// Mitsubishi GX Developer project: continuous   PLC: FX3U

PROGRAM MAIN
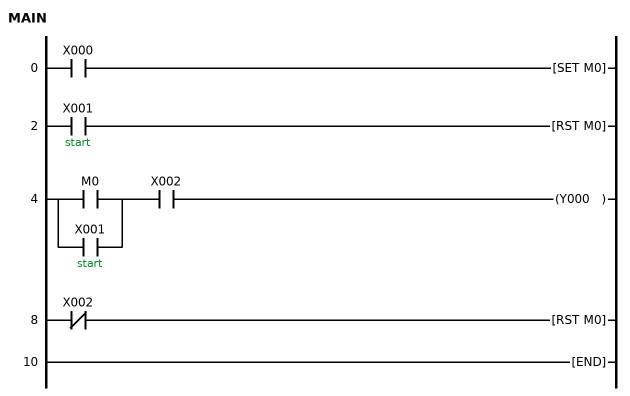
0     LD      X000
      SET     M0
2     LD      X001  ; start
      RST     M0
4     LD      M0
      OR      X001  ; start
      AND     X002
      OUT     Y000
8     LDI     X002
      RST     M0
10    END
END_PROGRAM
